// TIA Portal project "MarciaAvantiIndietro" (V20)

(* hardware
DEVICE "S7-1200 station_1"  S7-1200 Station
   slot 0: "Rack_0"  S7-1200 Rack  Rack  V1.0
   slot 1: "Playground_PLC"  CPU 1214C DC/DC/DC  6ES7 214-1AG40-0XB0  V4.7
   slot 3: "AQ 1x12BIT_1"  AQ1 signal board  6ES7 232-4HA30-0XB0  V1.0
*)

// ===== PLC "Playground_PLC"  CPU 1214C DC/DC/DC =====

VAR_GLOBAL   // PLC tag table "Default tag table"
   "AVANTI" AT %M0.0 : Bool;
   "INDIETRO" AT %M0.1 : Bool;
   "STOP" AT %M0.2 : Bool;
   "MARCIA_AVANTI" AT %M0.3 : Bool;
   "MARCIA_INDIETRO" AT %M0.4 : Bool;
   "START" AT %M0.5 : Bool;
   "SELETTORE_AVANTI" AT %M0.6 : Bool;
END_VAR

ORGANIZATION_BLOCK "Main"   // OB1, LAD, ProgramCycle
TITLE = "Main Program Sweep (Cycle)"
{ S7_Optimized_Access := 'TRUE' }
VERSION : 0.1
   VAR_INPUT
      Initial_Call : Bool;   // Initial call of this OB
      Remanence : Bool;   // =True, if remanent data are available
   END_VAR
   VAR_TEMP   // added for the SCL form of the ladder/FBD networks
      _w1 : Bool;
   END_VAR
BEGIN

REGION Network 1
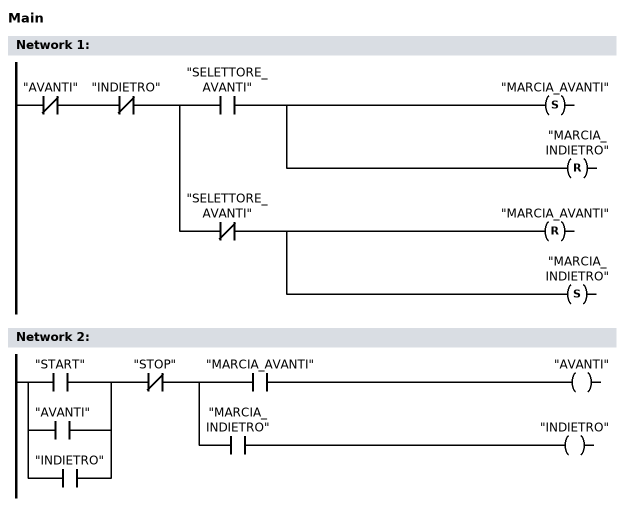
   RUNG wire#powerrail
      I_Contact( "AVANTI" )
      I_Contact( "INDIETRO" )
      wire#w1
      Contact( "SELETTORE_AVANTI" )
      wire#w2
      S_Coil( "MARCIA_AVANTI" )
   END_RUNG
   RUNG wire#w2
      R_Coil( "MARCIA_INDIETRO" )
   END_RUNG
   RUNG wire#w1
      I_Contact( "SELETTORE_AVANTI" )
      wire#w3
      R_Coil( "MARCIA_AVANTI" )
   END_RUNG
   RUNG wire#w3
      S_Coil( "MARCIA_INDIETRO" )
   END_RUNG
   // the same network as SCL:
   #_w1 := NOT "AVANTI" AND NOT "INDIETRO";
   IF #_w1 AND "SELETTORE_AVANTI" THEN
       "MARCIA_AVANTI" := TRUE;
       "MARCIA_INDIETRO" := FALSE;
   END_IF;
   IF #_w1 AND NOT "SELETTORE_AVANTI" THEN
       "MARCIA_AVANTI" := FALSE;
       "MARCIA_INDIETRO" := TRUE;
   END_IF;
END_REGION

REGION Network 2
   RUNG wire#powerrail
      Contact( "START" )
      wire#w1
      I_Contact( "STOP" )
      wire#w2
      Contact( "MARCIA_AVANTI" )
      Coil( "AVANTI" )
   END_RUNG
   RUNG wire#powerrail
      Contact( "AVANTI" )
   END_RUNG wire#w1
   RUNG wire#powerrail
      Contact( "INDIETRO" )
   END_RUNG wire#w1
   RUNG wire#w2
      Contact( "MARCIA_INDIETRO" )
      Coil( "INDIETRO" )
   END_RUNG
   // the same network as SCL:
   #_w1 := ("START" OR "AVANTI" OR "INDIETRO") AND NOT "STOP";
   "AVANTI" := #_w1 AND "MARCIA_AVANTI";
   "INDIETRO" := #_w1 AND "MARCIA_INDIETRO";
END_REGION
END_ORGANIZATION_BLOCK